// TIA Portal V17 export
// export: Created 2025-03-12T15:37:44.8789464Z, ExportSetting WithDefaults, DisplayName Totally Integrated Automation Portal, DisplayVersion V17 Update 8, DisplayName TIA Portal Openness, DisplayVersion V17 Update 8, DisplayName TIA Portal Version Control Interface, DisplayVersion V17, DisplayName SINAMICS Startdrive Advanced, DisplayVersion V17 SP2, DisplayName SINAMICS Startdrive G110M, G120, G120C, G120D, G120P, G115D, DisplayVersion V17 SP2, DisplayName SINAMICS Startdrive G130, G150, S120, S150, SINAMICS MV, S210, DisplayVersion V17 SP2, DisplayName STEP 7 Professional, DisplayVersion V17 Update 8, DisplayName SINUMERIK ONE STEP 7 Toolbox, DisplayVersion V17 Update 12, DisplayName SINUMERIK 840D sl STEP 7 Toolbox, DisplayVersion V17 Update 12, DisplayName STEP 7 Safety, DisplayVersion V17 Update 6, DisplayName WinCC Advanced, DisplayVersion V17 Update 8
TYPE "POWDER FEEDER HMI VALUES SETPOINTS"
// stored: IsFailsafeCompliant false
   STRUCT
      CarrierGasNominalLine1 : Real;
      CarrierGasNominalLine2 : Real;
      DiskSpeedNominalLine1 : Real;
      DiskSpeedNominalLine2 : Real;
      StirrerSpeedNominalLine1 : Real;
      StirrerSpeedNominalLine2 : Real;
      HopperTempNominalLine1 : Real;
      HopperTempNominalLine2 : Real;
      Spare8 : Real;
      Spare9 : Real;
      Spare10 : Real;
      Spare11 : Real;
      Spare12 : Real;
      Spare13 : Real;
      Spare14 : Real;
      Spare15 : Real;
   END_STRUCT;
END_TYPE
